TYPE ST_MOVER_SELECTOR_STATE :
STRUCT
  MoverIndex  : UINT;
  AxisId      : UDINT;
  State       : ST_MOVER_STATE;

  Info        : ST_MOVER_INFO;
END_STRUCT
END_TYPE

(* stored: Version 1.1.0.1, ProductVersion 3.1.4026.18
   DUT ST_MOVER_SELECTOR_STATE: Id {20425aad-d0dd-415d-af12-5aebe90b3dbe} *)
